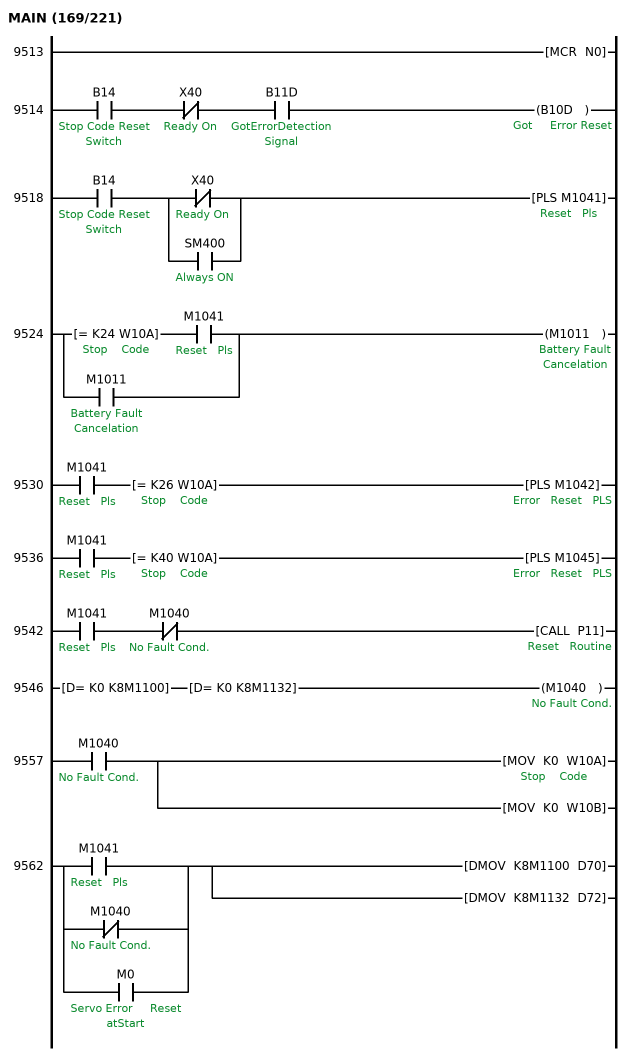
[picture p168: ladder of MAIN, rungs at steps 9513 to 9562]
9513  MCR     N0
9514  LD      B14  ; Stop Code Reset Switch
      ANI     X40  ; Ready On
      AND     B11D  ; GotErrorDetection Signal
      OUT     B10D  ; Got     Error Reset
9518  LD      B14  ; Stop Code Reset Switch
      LDI     X40  ; Ready On
      OR      SM400  ; Always ON
      ANB
      PLS     M1041  ; Reset   Pls
9524  LD=     K24 W10A  ; Stop    Code
      AND     M1041  ; Reset   Pls
      OR      M1011  ; Battery Fault   Cancelation
      OUT     M1011  ; Battery Fault   Cancelation
9530  LD      M1041  ; Reset   Pls
      AND=    K26 W10A  ; Stop    Code
      PLS     M1042  ; Error   Reset   PLS
9536  LD      M1041  ; Reset   Pls
      AND=    K40 W10A  ; Stop    Code
      PLS     M1045  ; Error   Reset   PLS
9542  LD      M1041  ; Reset   Pls
      ANI     M1040  ; No Fault Cond.
      CALL    P11  ; Reset   Routine
9546  LDD=    K0 K8M1100
      ANDD=   K0 K8M1132  ; Nozzle  Operation       Fault
      OUT     M1040  ; No Fault Cond.
9557  LD      M1040  ; No Fault Cond.
      MOV     K0 W10A
      MOV     K0 W10B
9562  LD      M1041  ; Reset   Pls
      ORI     M1040  ; No Fault Cond.
      OR      M0  ; Servo Error     Reset atStart
      DMOV    K8M1100 D70
      DMOV    K8M1132 D72
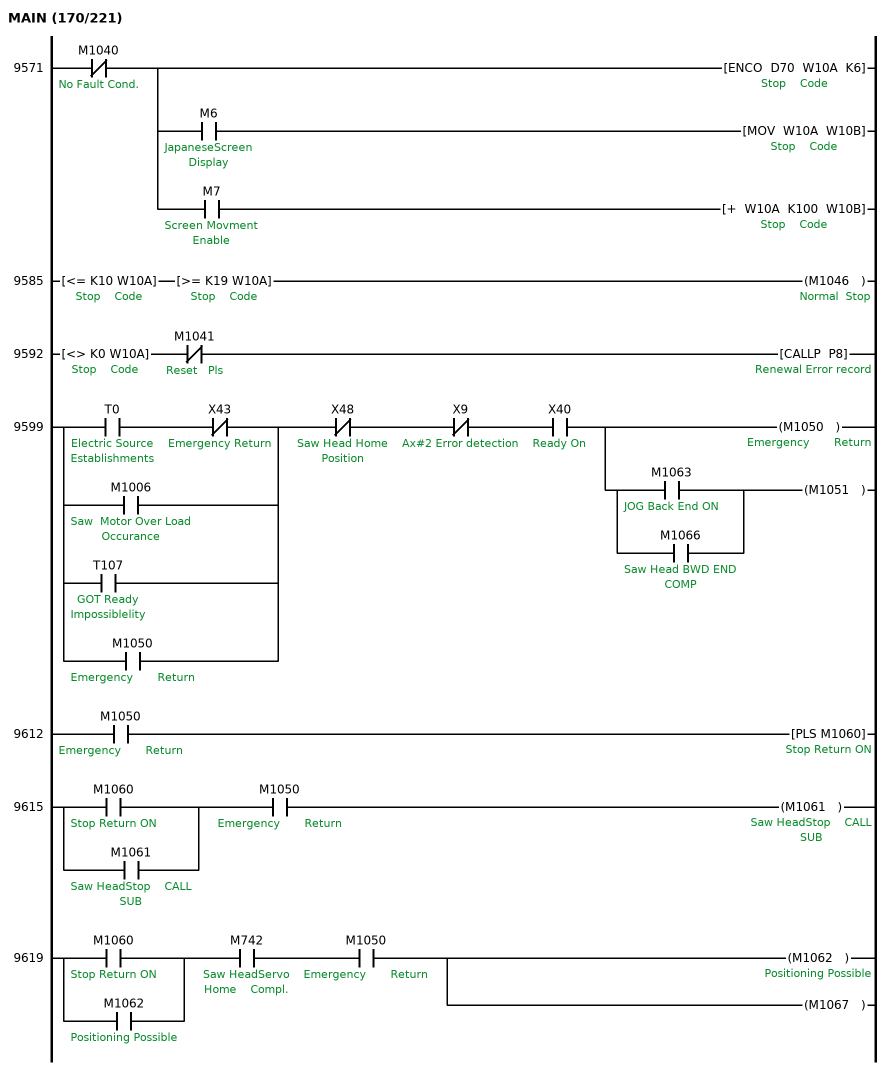
9571  LDI     M1040  ; No Fault Cond.
      ENCO    D70 W10A K6
      MPS
      AND     M6  ; JapaneseScreen Display
      MOV     W10A W10B
      MPP
      AND     M7  ; Screen Movment Enable
      +       W10A K100 W10B
9585  LD<=    K10 W10A  ; Stop    Code
      AND>=   K19 W10A  ; Stop    Code
      OUT     M1046  ; Normal  Stop
9592  LD<>    K0 W10A  ; Stop    Code
      ANI     M1041  ; Reset   Pls
      CALLP   P8  ; Renewal Error record
9599  LD      T0  ; Electric Source Establishments
      ANI     X43  ; Emergency Return
      OR      M1006  ; Saw  Motor Over Load Occurance
      OR      T107  ; GOT Ready Impossiblelity
      OR      M1050  ; Emergency       Return
      ANI     X48  ; Saw Head Home Position
      ANI     X9  ; Ax#2 Error detection
      AND     X40  ; Ready On
      OUT     M1050  ; Emergency       Return
      LD      M1063  ; JOG Back End ON
      OR      M1066  ; Saw Head BWD END COMP
      ANB
      OUT     M1051
9612  LD      M1050  ; Emergency       Return
      PLS     M1060  ; Stop Return ON
9615  LD      M1060  ; Stop Return ON
      OR      M1061  ; Saw HeadStop    CALL SUB
      AND     M1050  ; Emergency       Return
      OUT     M1061  ; Saw HeadStop    CALL SUB
9619  LD      M1060  ; Stop Return ON
      OR      M1062  ; Positioning Possible
      AND     M742  ; Saw HeadServo   Home    Compl.
      AND     M1050  ; Emergency       Return
      OUT     M1062  ; Positioning Possible
      OUT     M1067
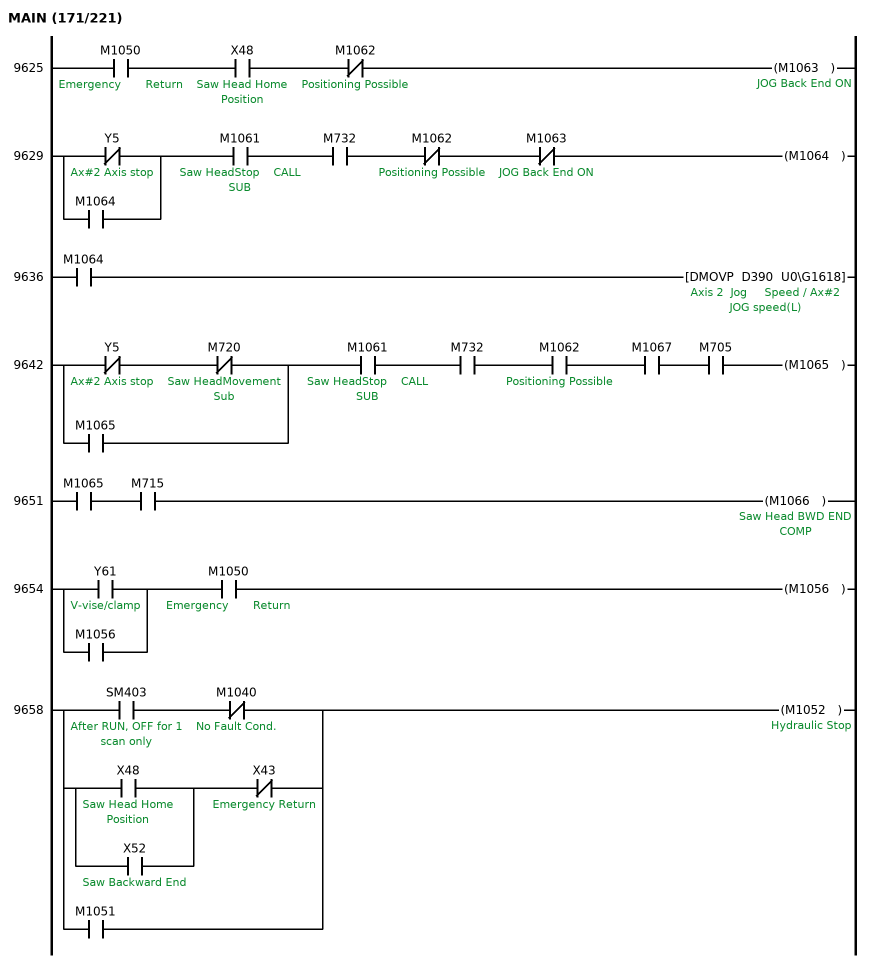
9625  LD      M1050  ; Emergency       Return
      AND     X48  ; Saw Head Home Position
      ANI     M1062  ; Positioning Possible
      OUT     M1063  ; JOG Back End ON
9629  LDI     Y5  ; Ax#2 Axis stop
      OR      M1064
      AND     M1061  ; Saw HeadStop    CALL SUB
      AND     M732
      ANI     M1062  ; Positioning Possible
      ANI     M1063  ; JOG Back End ON
      OUT     M1064
9636  LD      M1064
      DMOVP   D390 U0\G1618
9642  LDI     Y5  ; Ax#2 Axis stop
      ANI     M720  ; Saw HeadMovementSub
      OR      M1065
      AND     M1061  ; Saw HeadStop    CALL SUB
      AND     M732
      AND     M1062  ; Positioning Possible
      AND     M1067
      AND     M705
      OUT     M1065
9651  LD      M1065
      AND     M715
      OUT     M1066  ; Saw Head BWD END COMP
9654  LD      Y61  ; V-vise/clamp
      OR      M1056
      AND     M1050  ; Emergency       Return
      OUT     M1056
9658  LD      SM403  ; After RUN, OFF for 1 scan only
      ANI     M1040  ; No Fault Cond.
      LD      X48  ; Saw Head Home Position
      OR      X52  ; Saw Backward End
      ANI     X43  ; Emergency Return
      ORB
      OR      M1051
      OUT     M1052  ; Hydraulic Stop
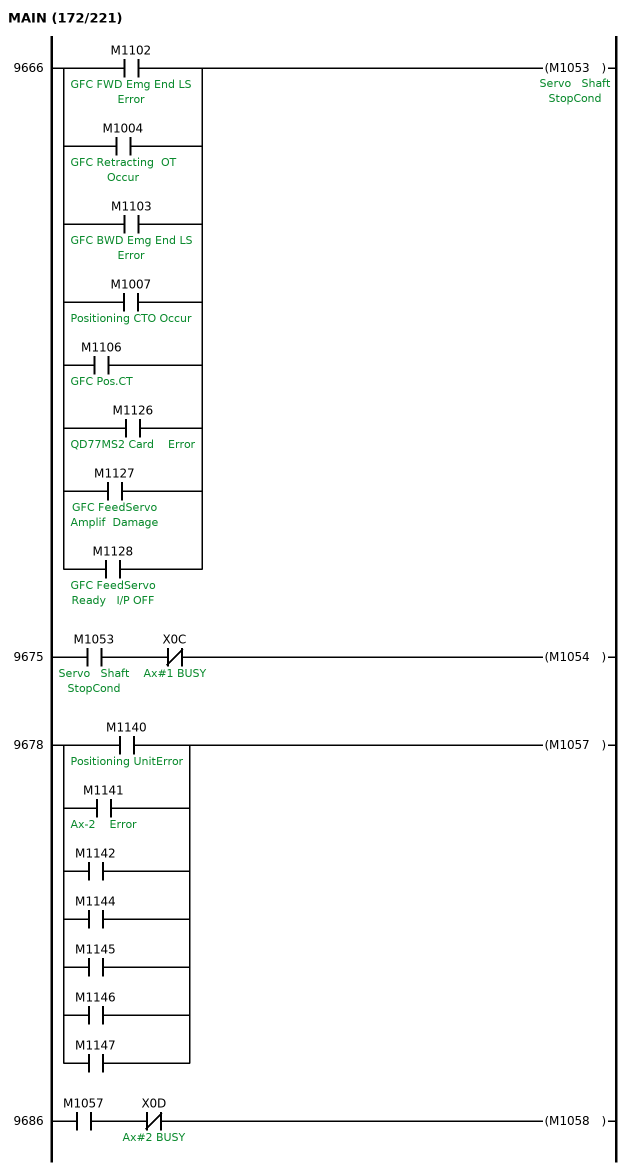
9666  LD      M1102  ; GFC FWD Emg End LS  Error
      OR      M1004  ; GFC Retracting  OT Occur
      OR      M1103  ; GFC BWD Emg End LS Error
      OR      M1007  ; Positioning CTO Occur
      OR      M1106  ; GFC Pos.CT
      OR      M1126  ; QD77MS2 Card    Error
      OR      M1127  ; GFC FeedServo   Amplif  Damage
      OR      M1128  ; GFC FeedServo   Ready   I/P OFF
      OUT     M1053  ; Servo   Shaft   StopCond
9675  LD      M1053  ; Servo   Shaft   StopCond
      ANI     X0C  ; Ax#1 BUSY
      OUT     M1054
9678  LD      M1140  ; Positioning UnitError
      OR      M1141  ; Ax-2    Error
      OR      M1142
      OR      M1144
      OR      M1145
      OR      M1146
      OR      M1147
      OUT     M1057
9686  LD      M1057
      ANI     X0D  ; Ax#2 BUSY
      OUT     M1058
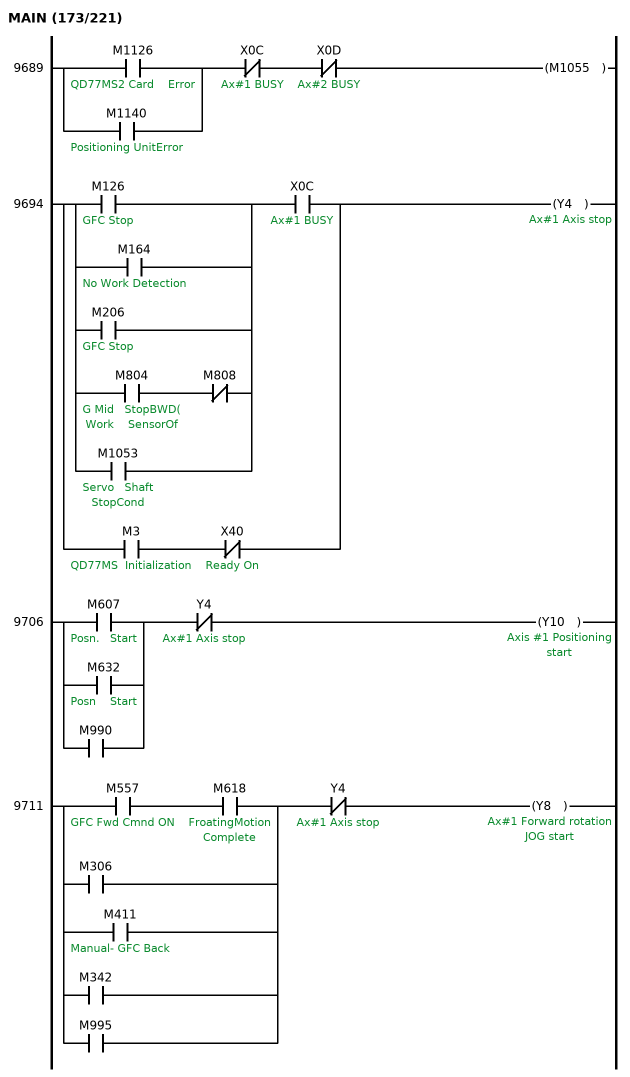
9689  LD      M1126  ; QD77MS2 Card    Error
      OR      M1140  ; Positioning UnitError
      ANI     X0C  ; Ax#1 BUSY
      ANI     X0D  ; Ax#2 BUSY
      OUT     M1055
9694  LD      M126  ; GFC Stop
      OR      M164  ; No Work Detection
      OR      M206  ; GFC Stop
      LD      M804  ; G Mid   StopBWD(Work    SensorOf
      ANI     M808
      ORB
      OR      M1053  ; Servo   Shaft   StopCond
      AND     X0C  ; Ax#1 BUSY
      LD      M3  ; QD77MS  Initialization
      ANI     X40  ; Ready On
      ORB
      OUT     Y4  ; Ax#1 Axis stop
9706  LD      M607  ; Posn.   Start
      OR      M632  ; Posn    Start
      OR      M990
      ANI     Y4  ; Ax#1 Axis stop
      OUT     Y10  ; Axis #1 Positioning start
9711  LD      M557  ; GFC Fwd Cmnd ON
      AND     M618  ; FroatingMotion  Complete
      OR      M306
      OR      M411  ; Manual- GFC Back
      OR      M342
      OR      M995
      ANI     Y4  ; Ax#1 Axis stop
      OUT     Y8  ; Ax#1 Forward rotation JOG start
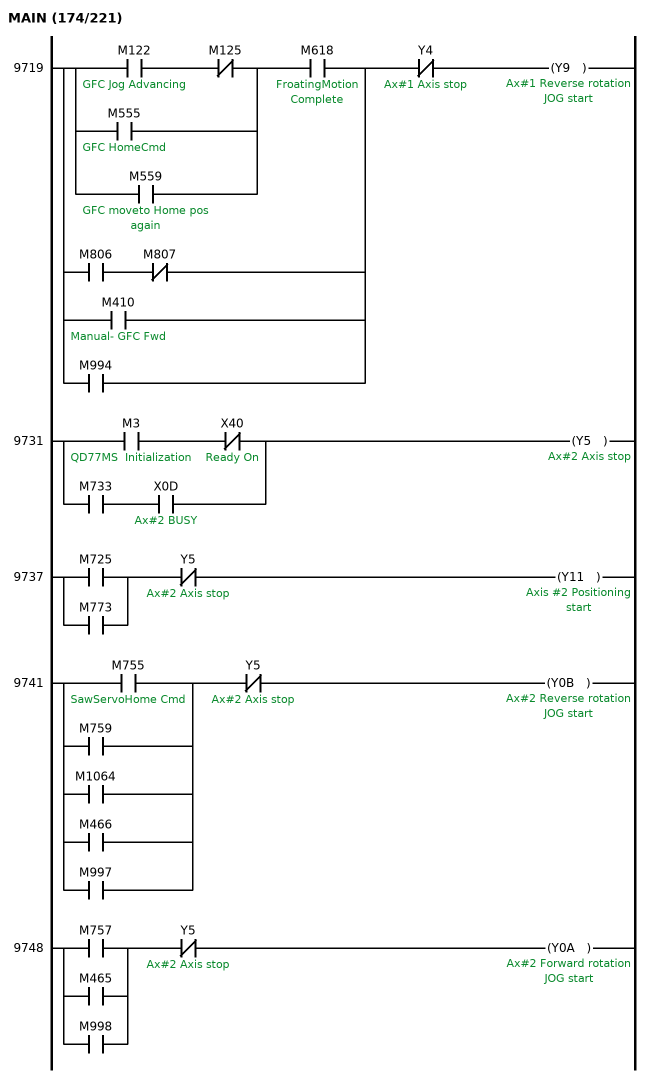
9719  LD      M122  ; GFC Jog Advancing
      ANI     M125
      OR      M555  ; GFC HomeCmd
      OR      M559  ; GFC moveto Home pos     again
      AND     M618  ; FroatingMotion  Complete
      LD      M806
      ANI     M807
      ORB
      OR      M410  ; Manual- GFC Fwd
      OR      M994
      ANI     Y4  ; Ax#1 Axis stop
      OUT     Y9  ; Ax#1 Reverse rotation JOG start
9731  LD      M3  ; QD77MS  Initialization
      ANI     X40  ; Ready On
      LD      M733
      AND     X0D  ; Ax#2 BUSY
      ORB
      OUT     Y5  ; Ax#2 Axis stop
9737  LD      M725
      OR      M773
      ANI     Y5  ; Ax#2 Axis stop
      OUT     Y11  ; Axis #2 Positioning start
9741  LD      M755  ; SawServoHome Cmd
      OR      M759
      OR      M1064
      OR      M466
      OR      M997
      ANI     Y5  ; Ax#2 Axis stop
      OUT     Y0B  ; Ax#2 Reverse rotation JOG start
9748  LD      M757
      OR      M465
      OR      M998
      ANI     Y5  ; Ax#2 Axis stop
      OUT     Y0A  ; Ax#2 Forward rotation JOG start
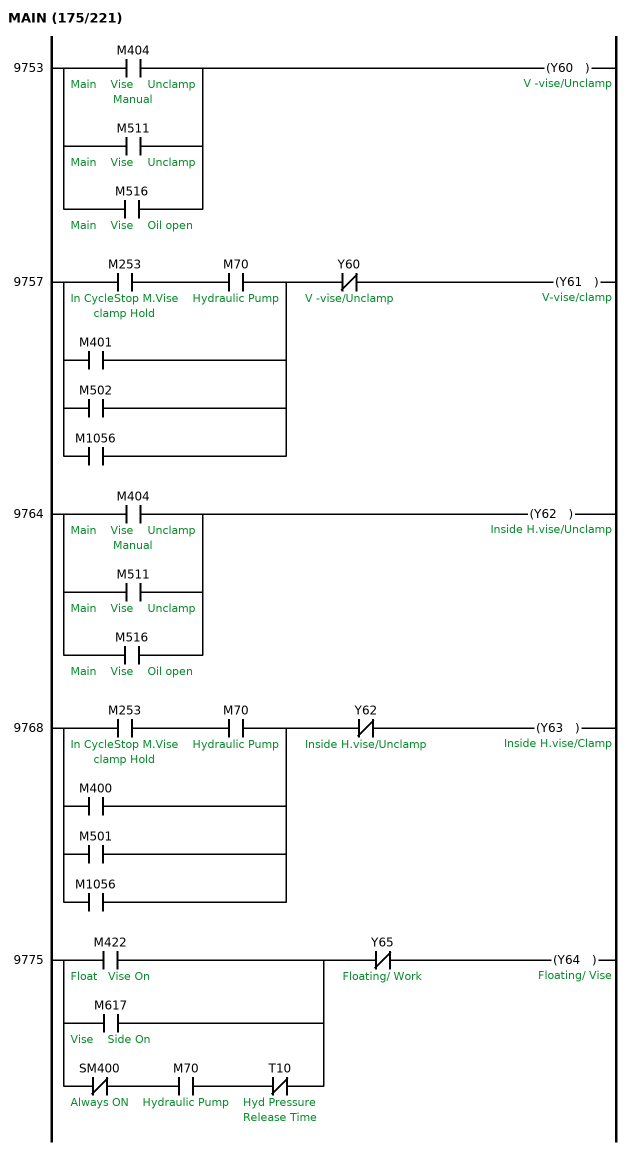
9753  LD      M404  ; Main    Vise    Unclamp Manual
      OR      M511  ; Main    Vise    Unclamp
      OR      M516  ; Main    Vise    Oil open
      OUT     Y60  ; V -vise/Unclamp
9757  LD      M253  ; In CycleStop M.Vise clamp Hold
      AND     M70  ; Hydraulic Pump
      OR      M401
      OR      M502
      OR      M1056
      ANI     Y60  ; V -vise/Unclamp
      OUT     Y61  ; V-vise/clamp
9764  LD      M404  ; Main    Vise    Unclamp Manual
      OR      M511  ; Main    Vise    Unclamp
      OR      M516  ; Main    Vise    Oil open
      OUT     Y62  ; Inside H.vise/Unclamp
9768  LD      M253  ; In CycleStop M.Vise clamp Hold
      AND     M70  ; Hydraulic Pump
      OR      M400
      OR      M501
      OR      M1056
      ANI     Y62  ; Inside H.vise/Unclamp
      OUT     Y63  ; Inside H.vise/Clamp
9775  LD      M422  ; Float   Vise On
      OR      M617  ; Vise    Side On
      LDI     SM400  ; Always ON
      AND     M70  ; Hydraulic Pump
      ANI     T10  ; Hyd Pressure    Release Time
      ORB
      ANI     Y65  ; Floating/ Work
      OUT     Y64  ; Floating/ Vise
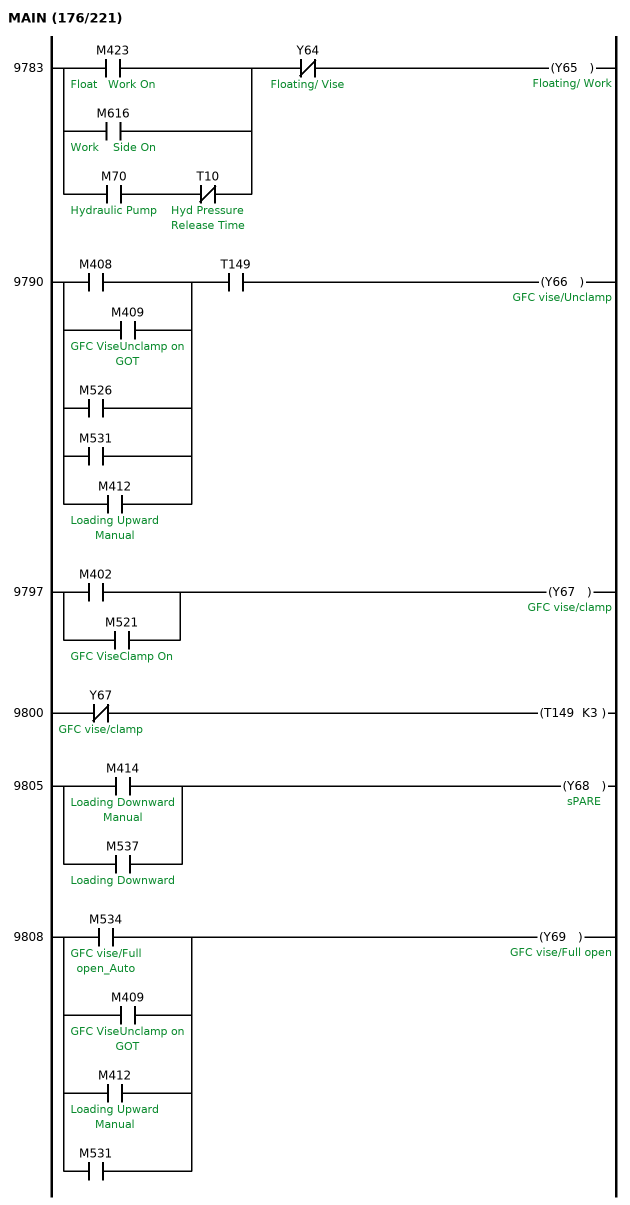
9783  LD      M423  ; Float   Work On
      OR      M616  ; Work    Side On
      LD      M70  ; Hydraulic Pump
      ANI     T10  ; Hyd Pressure    Release Time
      ORB
      ANI     Y64  ; Floating/ Vise
      OUT     Y65  ; Floating/ Work
9790  LD      M408
      OR      M409  ; GFC ViseUnclamp on GOT
      OR      M526
      OR      M531
      OR      M412  ; Loading Upward  Manual
      AND     T149
      OUT     Y66  ; GFC vise/Unclamp
9797  LD      M402
      OR      M521  ; GFC ViseClamp On
      OUT     Y67  ; GFC vise/clamp
9800  LDI     Y67  ; GFC vise/clamp
      OUT     T149 K3
9805  LD      M414  ; Loading Downward Manual
      OR      M537  ; Loading Downward
      OUT     Y68  ; sPARE
9808  LD      M534  ; GFC vise/Full open_Auto
      OR      M409  ; GFC ViseUnclamp on GOT
      OR      M412  ; Loading Upward  Manual
      OR      M531
      OUT     Y69  ; GFC vise/Full open
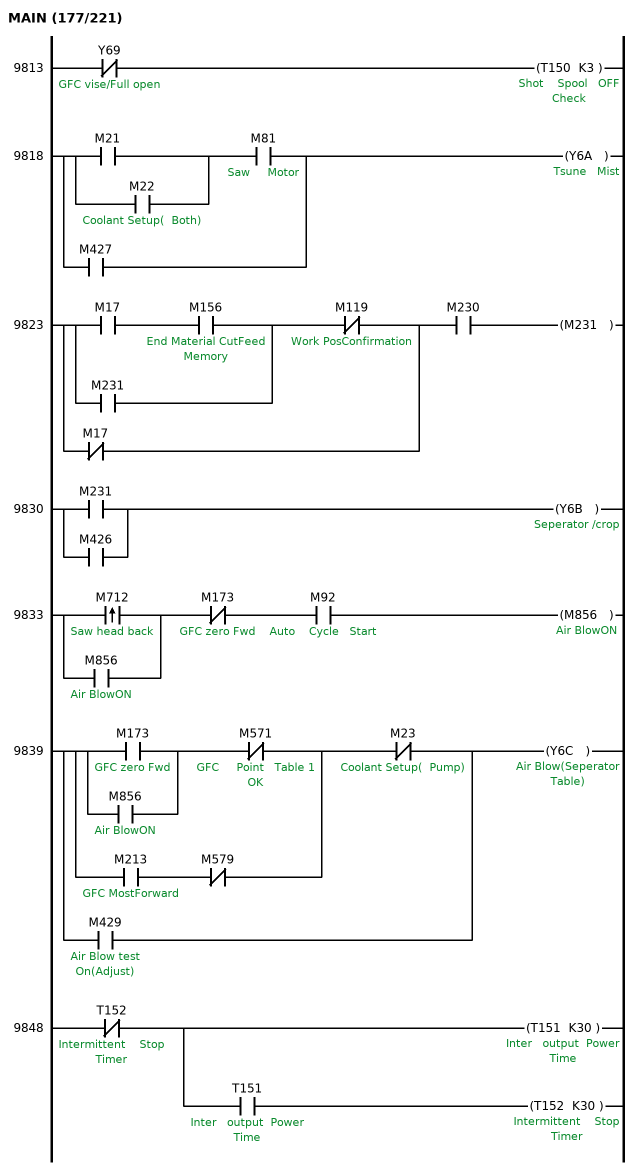
9813  LDI     Y69  ; GFC vise/Full open
      OUT     T150 K3  ; Shot    Spool   OFF     Check
9818  LD      M21
      OR      M22  ; Coolant Setup(  Both)
      AND     M81  ; Saw     Motor
      OR      M427
      OUT     Y6A  ; Tsune   Mist
9823  LD      M17
      AND     M156  ; End Material CutFeed Memory
      OR      M231
      ANI     M119  ; Work PosConfirmation
      ORI     M17
      AND     M230
      OUT     M231
9830  LD      M231
      OR      M426
      OUT     Y6B  ; Seperator /crop
9833  LDP     M712  ; Saw head back
      OR      M856  ; Air BlowON
      ANI     M173  ; GFC zero Fwd
      AND     M92  ; Auto    Cycle   Start
      OUT     M856  ; Air BlowON
9839  LD      M173  ; GFC zero Fwd
      OR      M856  ; Air BlowON
      ANI     M571  ; GFC     Point   Table 1 OK
      LD      M213  ; GFC MostForward
      ANI     M579
      ORB
      ANI     M23  ; Coolant Setup(  Pump)
      OR      M429  ; Air Blow test On(Adjust)
      OUT     Y6C  ; Air Blow(Seperator Table)
9848  LDI     T152  ; Intermittent    Stop    Timer
      OUT     T151 K30  ; Inter   output  Power   Time
      AND     T151  ; Inter   output  Power   Time
      OUT     T152 K30  ; Intermittent    Stop    Timer
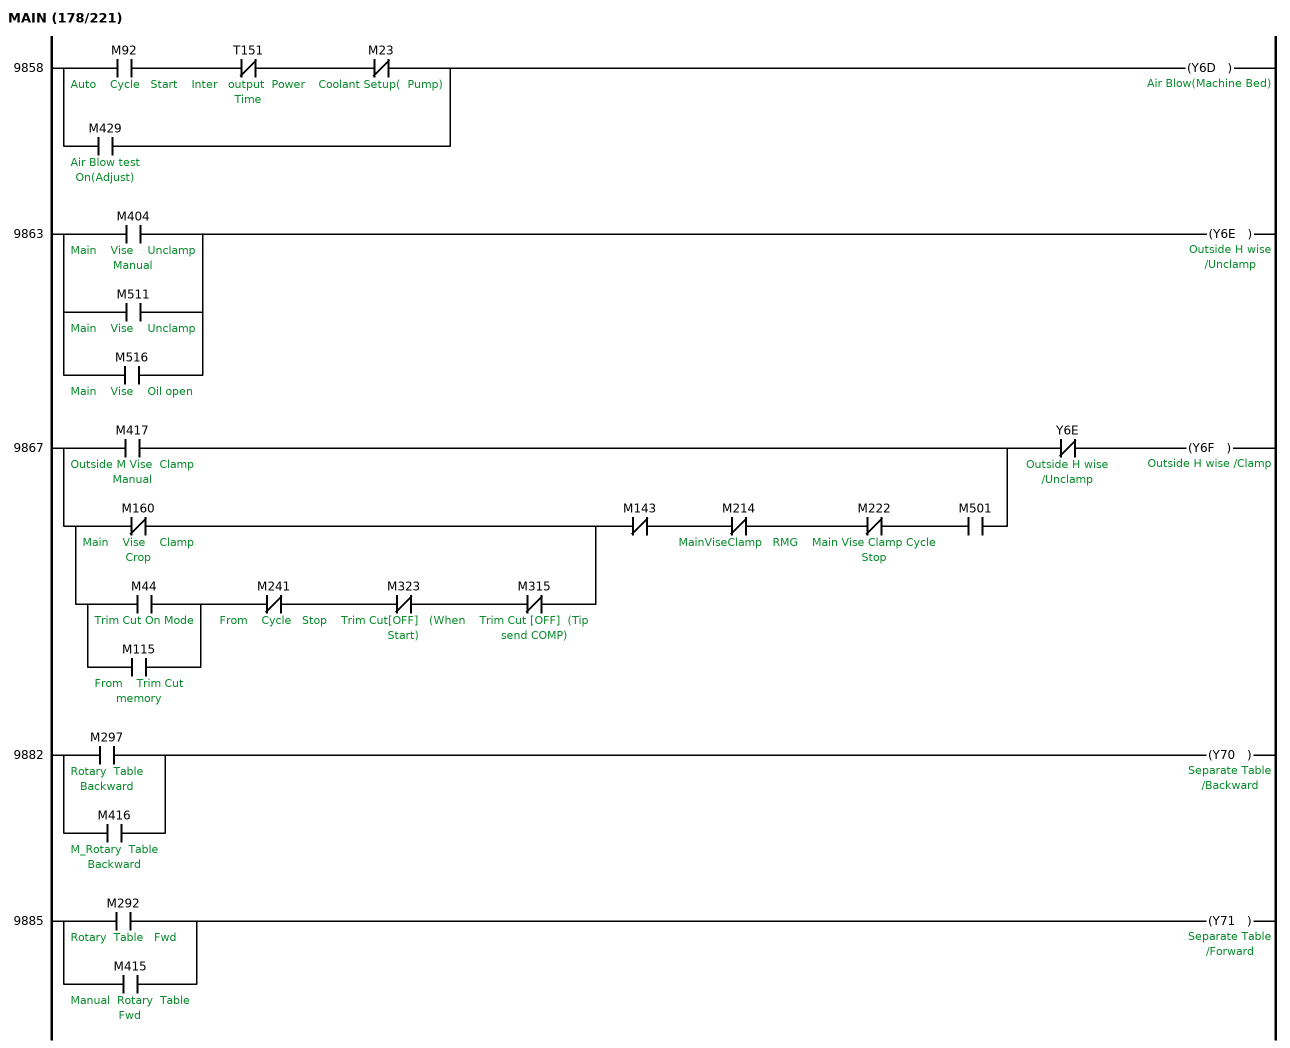
9858  LD      M92  ; Auto    Cycle   Start
      ANI     T151  ; Inter   output  Power   Time
      ANI     M23  ; Coolant Setup(  Pump)
      OR      M429  ; Air Blow test On(Adjust)
      OUT     Y6D  ; Air Blow(Machine Bed)
9863  LD      M404  ; Main    Vise    Unclamp Manual
      OR      M511  ; Main    Vise    Unclamp
      OR      M516  ; Main    Vise    Oil open
      OUT     Y6E  ; Outside H wise /Unclamp
9867  LD      M417  ; Outside M Vise  Clamp   Manual
      LDI     M160  ; Main    Vise    Clamp   Crop
      LD      M44  ; Trim Cut On Mode
      OR      M115  ; From    Trim Cut memory
      ANI     M241  ; From    Cycle   Stop
      ANI     M323  ; Trim Cut[OFF]   (When   Start)
      ANI     M315  ; Trim Cut [OFF]  (Tip send COMP)
      ORB
      ANI     M143
      ANI     M214  ; MainViseClamp   RMG
      ANI     M222  ; Main Vise Clamp Cycle Stop
      AND     M501
      ORB
      ANI     Y6E  ; Outside H wise /Unclamp
      OUT     Y6F  ; Outside H wise /Clamp
9882  LD      M297  ; Rotary  Table   Backward
      OR      M416  ; M_Rotary  Table Backward
      OUT     Y70  ; Separate Table /Backward
9885  LD      M292  ; Rotary  Table   Fwd
      OR      M415  ; Manual  Rotary  Table   Fwd
      OUT     Y71  ; Separate Table /Forward
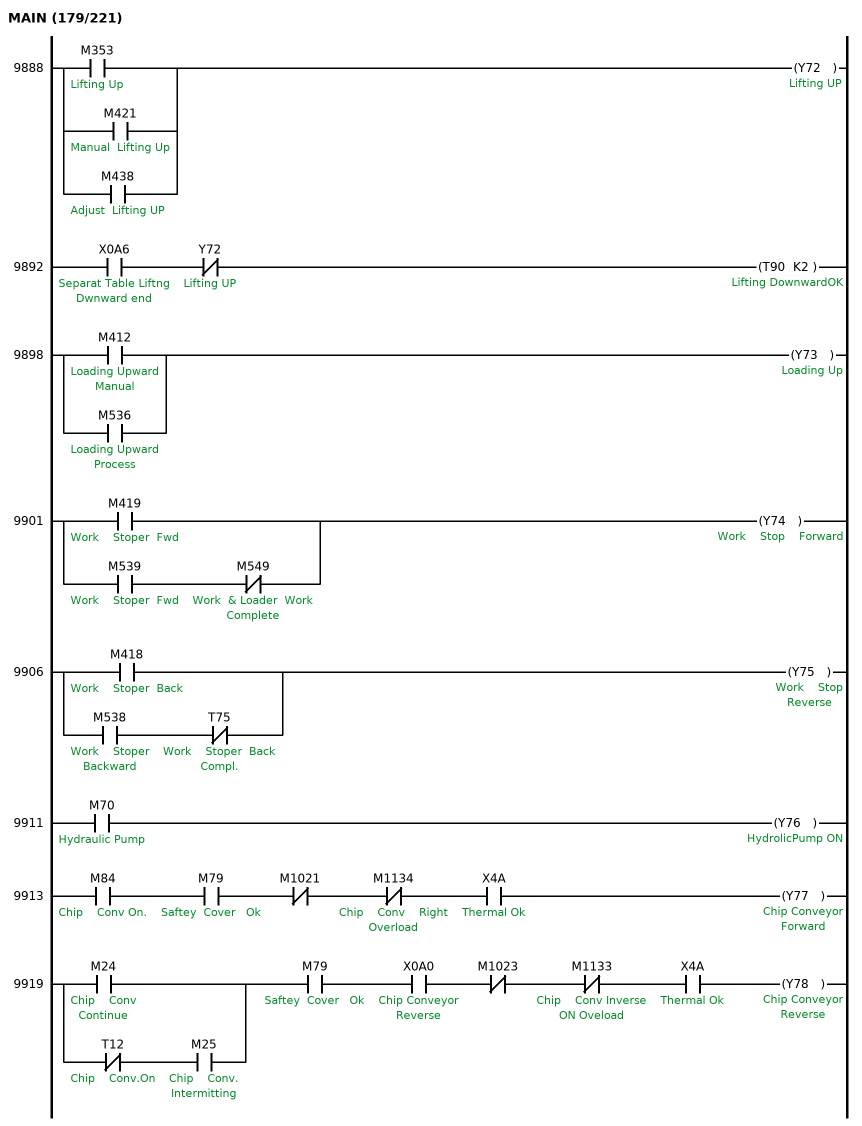
9888  LD      M353  ; Lifting Up
      OR      M421  ; Manual  Lifting Up
      OR      M438  ; Adjust  Lifting UP
      OUT     Y72  ; Lifting UP
9892  LD      X0A6  ; Separat Table Liftng Dwnward end
      ANI     Y72  ; Lifting UP
      OUT     T90 K2  ; Lifting DownwardOK
9898  LD      M412  ; Loading Upward  Manual
      OR      M536  ; Loading Upward  Process
      OUT     Y73  ; Loading Up
9901  LD      M419  ; Work    Stoper  Fwd
      LD      M539  ; Work    Stoper  Fwd
      ANI     M549  ; Work  & Loader  Work Complete
      ORB
      OUT     Y74  ; Work    Stop    Forward
9906  LD      M418  ; Work    Stoper  Back
      LD      M538  ; Work    Stoper  Backward
      ANI     T75  ; Work    Stoper  Back    Compl.
      ORB
      OUT     Y75  ; Work    Stop    Reverse
9911  LD      M70  ; Hydraulic Pump
      OUT     Y76  ; HydrolicPump ON
9913  LD      M84  ; Chip    Conv On.
      AND     M79  ; Saftey  Cover   Ok
      ANI     M1021
      ANI     M1134  ; Chip    Conv    Right   Overload
      AND     X4A  ; Thermal Ok
      OUT     Y77  ; Chip Conveyor Forward
9919  LD      M24  ; Chip    Conv    Continue
      LDI     T12  ; Chip    Conv.On
      AND     M25  ; Chip    Conv.   Intermitting
      ORB
      AND     M79  ; Saftey  Cover   Ok
      AND     X0A0  ; Chip Conveyor Reverse
      ANI     M1023
      ANI     M1133  ; Chip    Conv Inverse ON Oveload
      AND     X4A  ; Thermal Ok
      OUT     Y78  ; Chip Conveyor Reverse
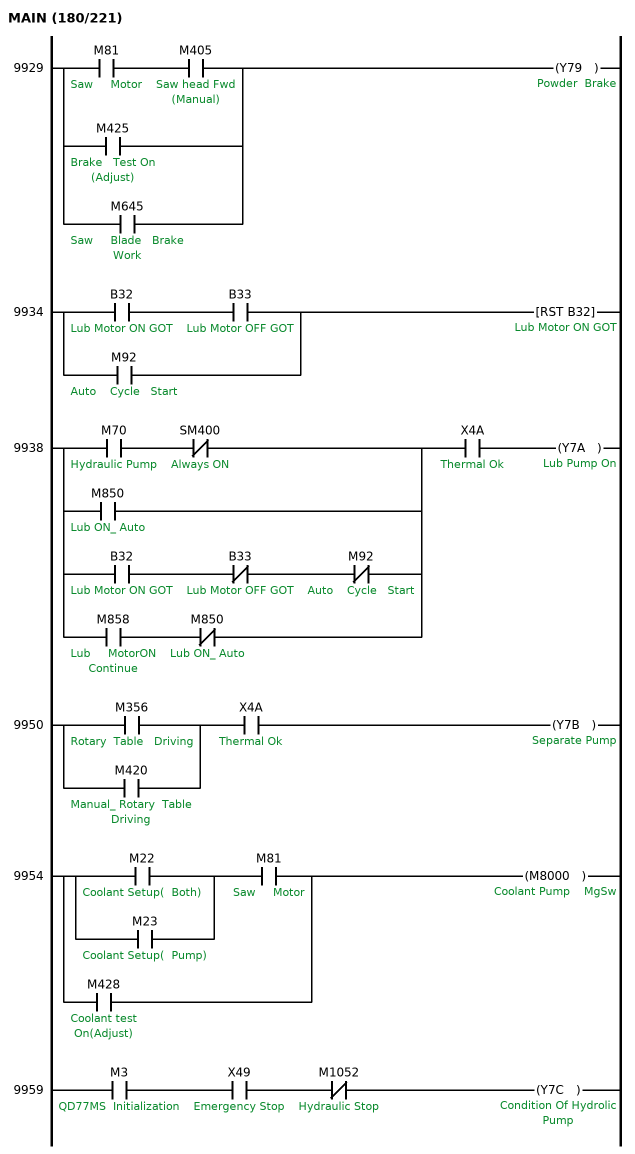
9929  LD      M81  ; Saw     Motor
      AND     M405  ; Saw head Fwd    (Manual)
      OR      M425  ; Brake   Test On (Adjust)
      OR      M645  ; Saw     Blade   Brake   Work
      OUT     Y79  ; Powder  Brake
9934  LD      B32  ; Lub Motor ON GOT
      AND     B33  ; Lub Motor OFF GOT
      OR      M92  ; Auto    Cycle   Start
      RST     B32  ; Lub Motor ON GOT
9938  LD      M70  ; Hydraulic Pump
      ANI     SM400  ; Always ON
      OR      M850  ; Lub ON_ Auto
      LD      B32  ; Lub Motor ON GOT
      ANI     B33  ; Lub Motor OFF GOT
      ANI     M92  ; Auto    Cycle   Start
      ORB
      LD      M858  ; Lub     MotorON Continue
      ANI     M850  ; Lub ON_ Auto
      ORB
      AND     X4A  ; Thermal Ok
      OUT     Y7A  ; Lub Pump On
9950  LD      M356  ; Rotary  Table   Driving
      OR      M420  ; Manual_ Rotary  Table   Driving
      AND     X4A  ; Thermal Ok
      OUT     Y7B  ; Separate Pump
9954  LD      M22  ; Coolant Setup(  Both)
      OR      M23  ; Coolant Setup(  Pump)
      AND     M81  ; Saw     Motor
      OR      M428  ; Coolant test On(Adjust)
      OUT     M8000  ; Coolant Pump    MgSw
9959  LD      M3  ; QD77MS  Initialization
      AND     X49  ; Emergency Stop
      ANI     M1052  ; Hydraulic Stop
      OUT     Y7C  ; Condition Of Hydrolic Pump
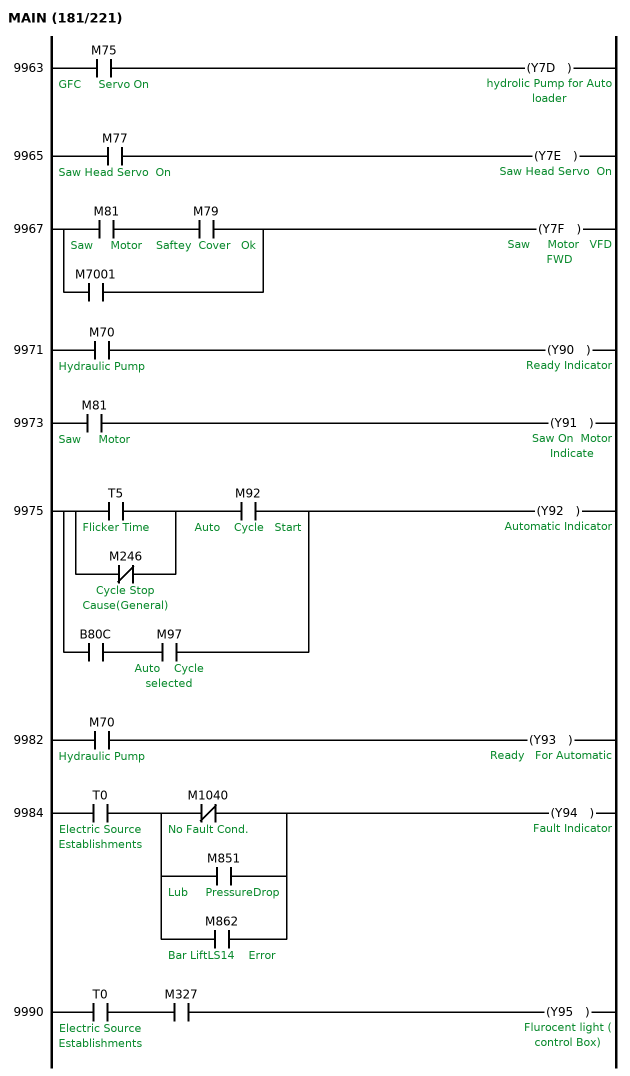
9963  LD      M75  ; GFC     Servo On
      OUT     Y7D  ; hydrolic Pump for Auto loader
9965  LD      M77  ; Saw Head Servo  On
      OUT     Y7E  ; Saw Head Servo  On
9967  LD      M81  ; Saw     Motor
      AND     M79  ; Saftey  Cover   Ok
      OR      M7001
      OUT     Y7F  ; Saw     Motor   VFD FWD
9971  LD      M70  ; Hydraulic Pump
      OUT     Y90  ; Ready Indicator
9973  LD      M81  ; Saw     Motor
      OUT     Y91  ; Saw On  Motor   Indicate
9975  LD      T5  ; Flicker Time
      ORI     M246  ; Cycle Stop Cause(General)
      AND     M92  ; Auto    Cycle   Start
      LD      B80C
      AND     M97  ; Auto    Cycle   selected
      ORB
      OUT     Y92  ; Automatic Indicator
9982  LD      M70  ; Hydraulic Pump
      OUT     Y93  ; Ready   For Automatic
9984  LD      T0  ; Electric Source Establishments
      LDI     M1040  ; No Fault Cond.
      OR      M851  ; Lub     PressureDrop
      OR      M862  ; Bar LiftLS14    Error
      ANB
      OUT     Y94  ; Fault Indicator
9990  LD      T0  ; Electric Source Establishments
      AND     M327
      OUT     Y95  ; Flurocent light ( control Box)
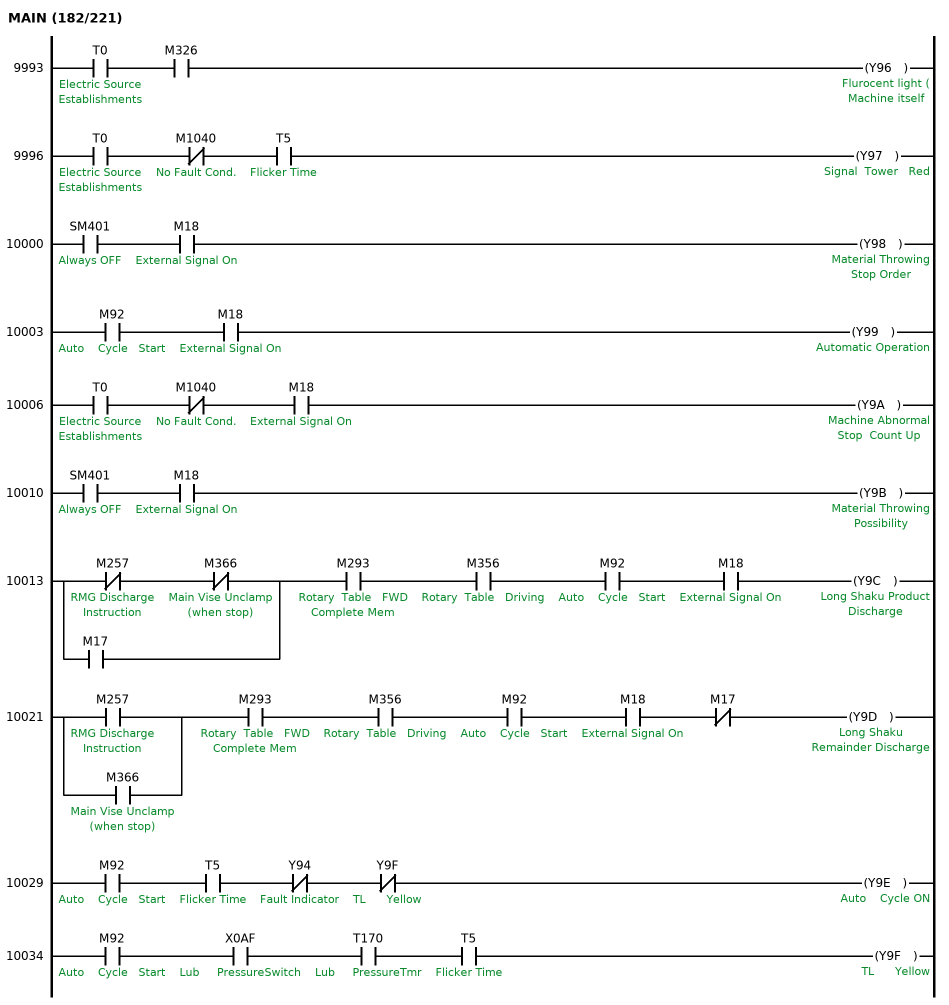
9993  LD      T0  ; Electric Source Establishments
      AND     M326
      OUT     Y96  ; Flurocent light ( Machine itself
9996  LD      T0  ; Electric Source Establishments
      ANI     M1040  ; No Fault Cond.
      AND     T5  ; Flicker Time
      OUT     Y97  ; Signal  Tower   Red
10000 LD      SM401  ; Always OFF
      AND     M18  ; External Signal On
      OUT     Y98  ; Material Throwing Stop Order
10003 LD      M92  ; Auto    Cycle   Start
      AND     M18  ; External Signal On
      OUT     Y99  ; Automatic Operation
10006 LD      T0  ; Electric Source Establishments
      ANI     M1040  ; No Fault Cond.
      AND     M18  ; External Signal On
      OUT     Y9A  ; Machine Abnormal Stop  Count Up
10010 LD      SM401  ; Always OFF
      AND     M18  ; External Signal On
      OUT     Y9B  ; Material Throwing Possibility
10013 LDI     M257  ; RMG Discharge Instruction
      ANI     M366  ; Main Vise Unclamp (when stop)
      OR      M17
      AND     M293  ; Rotary  Table   FWD Complete Mem
      AND     M356  ; Rotary  Table   Driving
      AND     M92  ; Auto    Cycle   Start
      AND     M18  ; External Signal On
      OUT     Y9C  ; Long Shaku Product Discharge
10021 LD      M257  ; RMG Discharge Instruction
      OR      M366  ; Main Vise Unclamp (when stop)
      AND     M293  ; Rotary  Table   FWD Complete Mem
      AND     M356  ; Rotary  Table   Driving
      AND     M92  ; Auto    Cycle   Start
      AND     M18  ; External Signal On
      ANI     M17
      OUT     Y9D  ; Long Shaku Remainder Discharge
10029 LD      M92  ; Auto    Cycle   Start
      AND     T5  ; Flicker Time
      ANI     Y94  ; Fault Indicator
      ANI     Y9F  ; TL      Yellow
      OUT     Y9E  ; Auto    Cycle ON
10034 LD      M92  ; Auto    Cycle   Start
      AND     X0AF  ; Lub     PressureSwitch
      AND     T170  ; Lub     PressureTmr
      AND     T5  ; Flicker Time
      OUT     Y9F  ; TL      Yellow
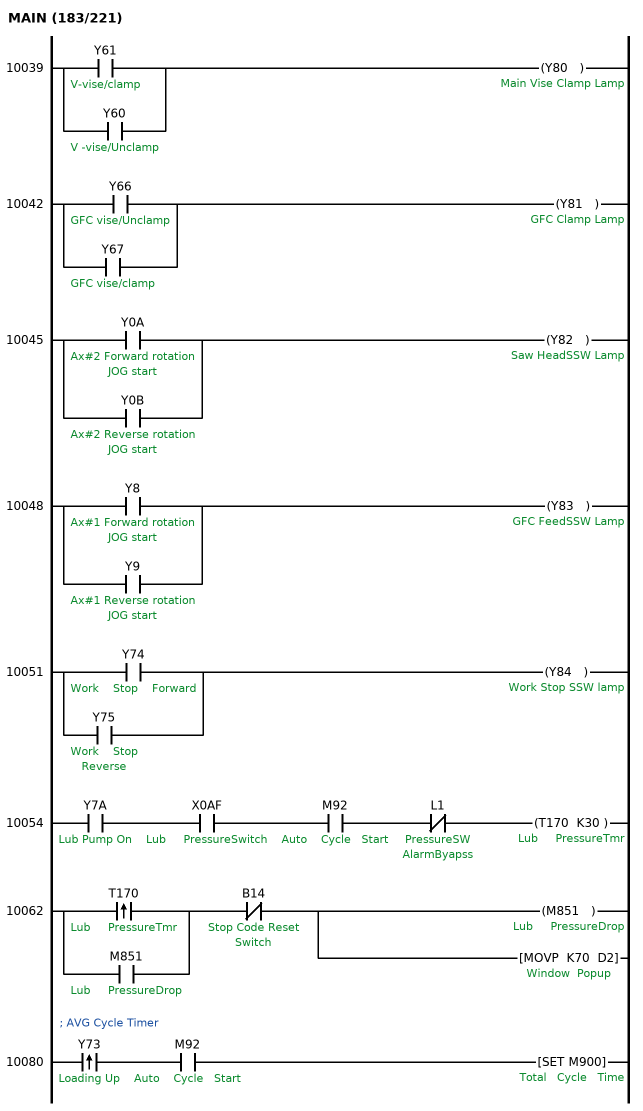
10039 LD      Y61  ; V-vise/clamp
      OR      Y60  ; V -vise/Unclamp
      OUT     Y80  ; Main Vise Clamp Lamp
10042 LD      Y66  ; GFC vise/Unclamp
      OR      Y67  ; GFC vise/clamp
      OUT     Y81  ; GFC Clamp Lamp
10045 LD      Y0A  ; Ax#2 Forward rotation JOG start
      OR      Y0B  ; Ax#2 Reverse rotation JOG start
      OUT     Y82  ; Saw HeadSSW Lamp
10048 LD      Y8  ; Ax#1 Forward rotation JOG start
      OR      Y9  ; Ax#1 Reverse rotation JOG start
      OUT     Y83  ; GFC FeedSSW Lamp
10051 LD      Y74  ; Work    Stop    Forward
      OR      Y75  ; Work    Stop    Reverse
      OUT     Y84  ; Work Stop SSW lamp
10054 LD      Y7A  ; Lub Pump On
      AND     X0AF  ; Lub     PressureSwitch
      AND     M92  ; Auto    Cycle   Start
      ANI     L1  ; PressureSW AlarmByapss
      OUT     T170 K30  ; Lub     PressureTmr
10062 LDP     T170  ; Lub     PressureTmr
      OR      M851  ; Lub     PressureDrop
      ANI     B14  ; Stop Code Reset Switch
      OUT     M851  ; Lub     PressureDrop
      MOVP    K70 D2
; AVG Cycle Timer
10080 LDP     Y73  ; Loading Up
      AND     M92  ; Auto    Cycle   Start
      SET     M900  ; Total   Cycle   Time
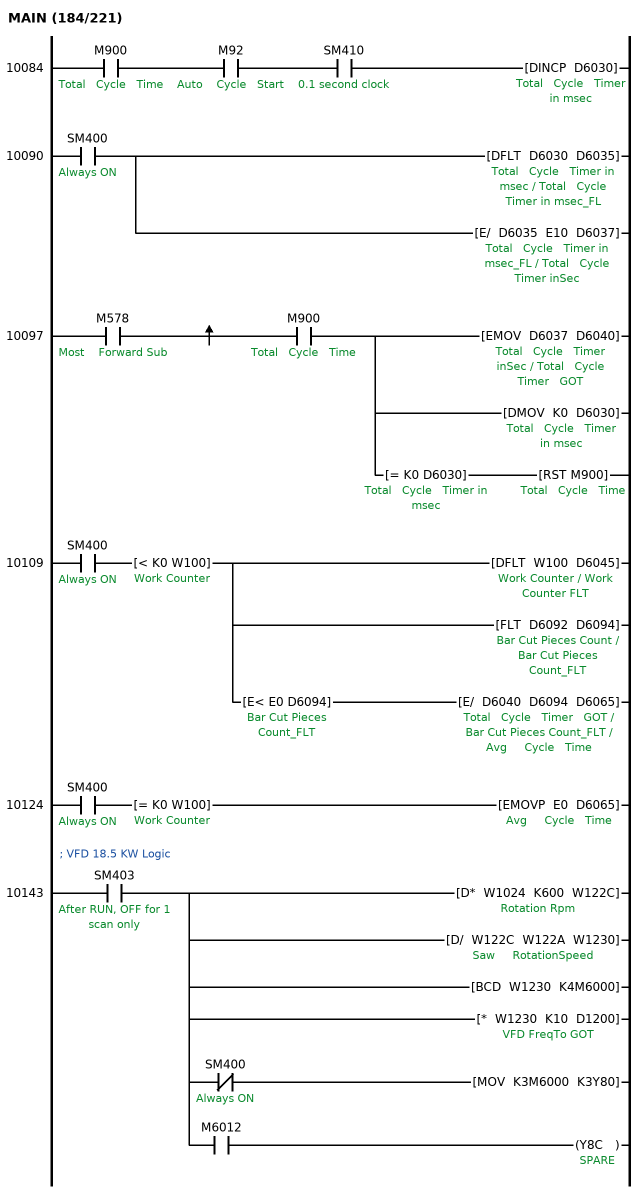
10084 LD      M900  ; Total   Cycle   Time
      AND     M92  ; Auto    Cycle   Start
      AND     SM410  ; 0.1 second clock
      DINCP   D6030  ; Total   Cycle   Timer in msec
10090 LD      SM400  ; Always ON
      DFLT    D6030 D6035  ; Total   Cycle   Timer in msec_FL
      E/      D6035 E10 D6037  ; Total   Cycle   Timer inSec
10097 LD      M578  ; Most    Forward Sub
      MEP
      AND     M900  ; Total   Cycle   Time
      EMOV    D6037 D6040  ; Total   Cycle   Timer   GOT
      DMOV    K0 D6030
      AND=    K0 D6030  ; Total   Cycle   Timer in msec
      RST     M900  ; Total   Cycle   Time
10109 LD      SM400  ; Always ON
      AND<    K0 W100  ; Work Counter
      DFLT    W100 D6045  ; Work    Counter FLT
      FLT     D6092 D6094  ; Bar Cut Pieces Count_FLT
      ANDE<   E0 D6094  ; Bar Cut Pieces Count_FLT
      E/      D6040 D6094 D6065  ; Avg     Cycle   Time
10124 LD      SM400  ; Always ON
      AND=    K0 W100  ; Work Counter
      EMOVP   E0 D6065
; VFD 18.5 KW Logic
10143 LD      SM403  ; After RUN, OFF for 1 scan only
      D*      W1024 K600 W122C
      D/      W122C W122A W1230  ; Saw     RotationSpeed
      BCD     W1230 K4M6000
      *       W1230 K10 D1200  ; VFD FreqTo GOT
      MPS
      ANI     SM400  ; Always ON
      MOV     K3M6000 K3Y80
      MPP
      AND     M6012
      OUT     Y8C  ; SPARE
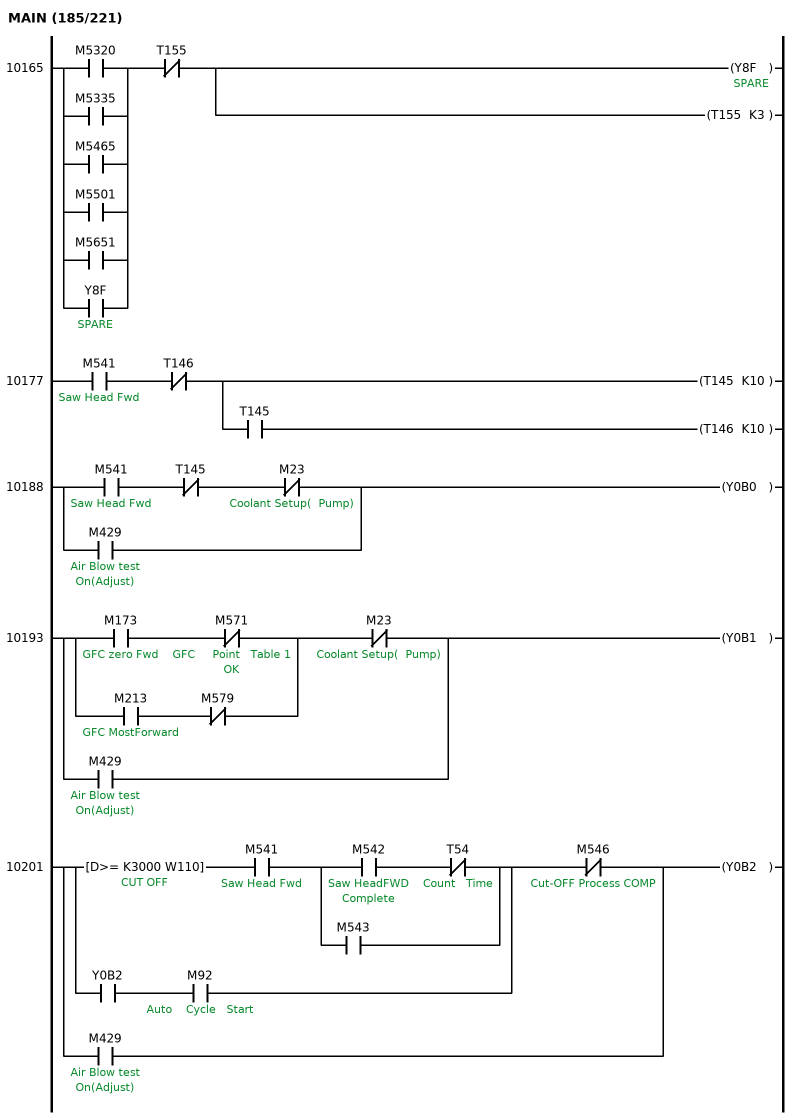
10165 LD      M5320
      OR      M5335
      OR      M5465
      OR      M5501
      OR      M5651
      OR      Y8F  ; SPARE
      ANI     T155
      OUT     Y8F  ; SPARE
      OUT     T155 K3
10177 LD      M541  ; Saw Head Fwd
      ANI     T146
      OUT     T145 K10
      AND     T145
      OUT     T146 K10
10188 LD      M541  ; Saw Head Fwd
      ANI     T145
      ANI     M23  ; Coolant Setup(  Pump)
      OR      M429  ; Air Blow test On(Adjust)
      OUT     Y0B0
10193 LD      M173  ; GFC zero Fwd
      ANI     M571  ; GFC     Point   Table 1 OK
      LD      M213  ; GFC MostForward
      ANI     M579
      ORB
      ANI     M23  ; Coolant Setup(  Pump)
      OR      M429  ; Air Blow test On(Adjust)
      OUT     Y0B1
10201 LDD>=   K3000 W110  ; CUT OFF
      AND     M541  ; Saw Head Fwd
      LD      M542  ; Saw HeadFWD     Complete
      ANI     T54  ; Count   Time
      OR      M543
      ANB
      LD      Y0B2
      AND     M92  ; Auto    Cycle   Start
      ORB
      ANI     M546  ; Cut-OFF Process COMP
      OR      M429  ; Air Blow test On(Adjust)
      OUT     Y0B2
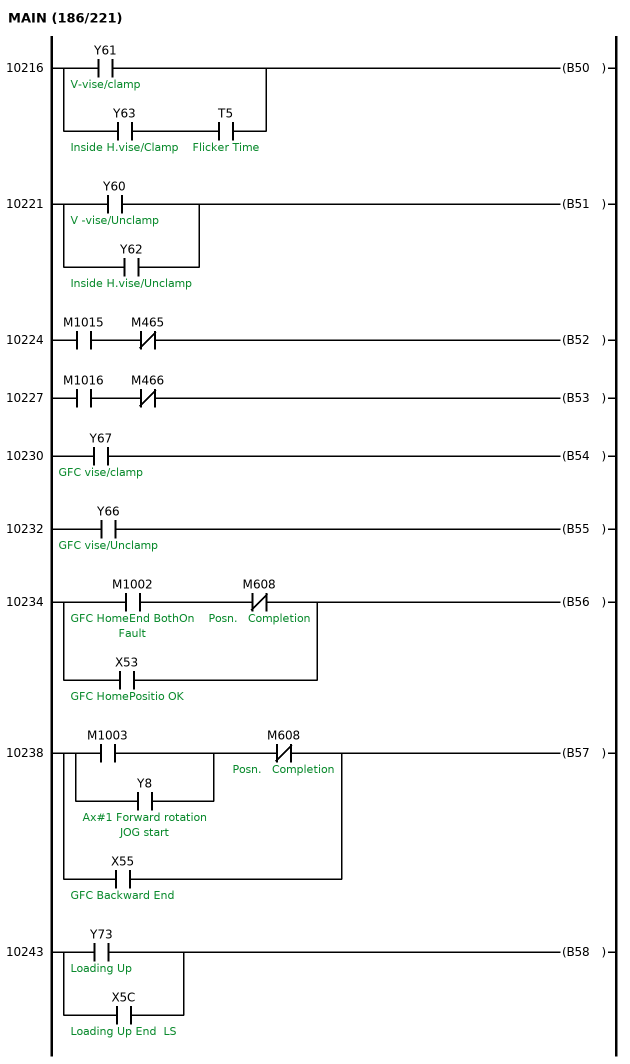
10216 LD      Y61  ; V-vise/clamp
      LD      Y63  ; Inside H.vise/Clamp
      AND     T5  ; Flicker Time
      ORB
      OUT     B50
10221 LD      Y60  ; V -vise/Unclamp
      OR      Y62  ; Inside H.vise/Unclamp
      OUT     B51
10224 LD      M1015
      ANI     M465
      OUT     B52
10227 LD      M1016
      ANI     M466
      OUT     B53
10230 LD      Y67  ; GFC vise/clamp
      OUT     B54
10232 LD      Y66  ; GFC vise/Unclamp
      OUT     B55
10234 LD      M1002  ; GFC HomeEnd BothOn Fault
      ANI     M608  ; Posn.   Completion
      OR      X53  ; GFC HomePositio OK
      OUT     B56
10238 LD      M1003
      OR      Y8  ; Ax#1 Forward rotation JOG start
      ANI     M608  ; Posn.   Completion
      OR      X55  ; GFC Backward End
      OUT     B57
10243 LD      Y73  ; Loading Up
      OR      X5C  ; Loading Up End  LS
      OUT     B58
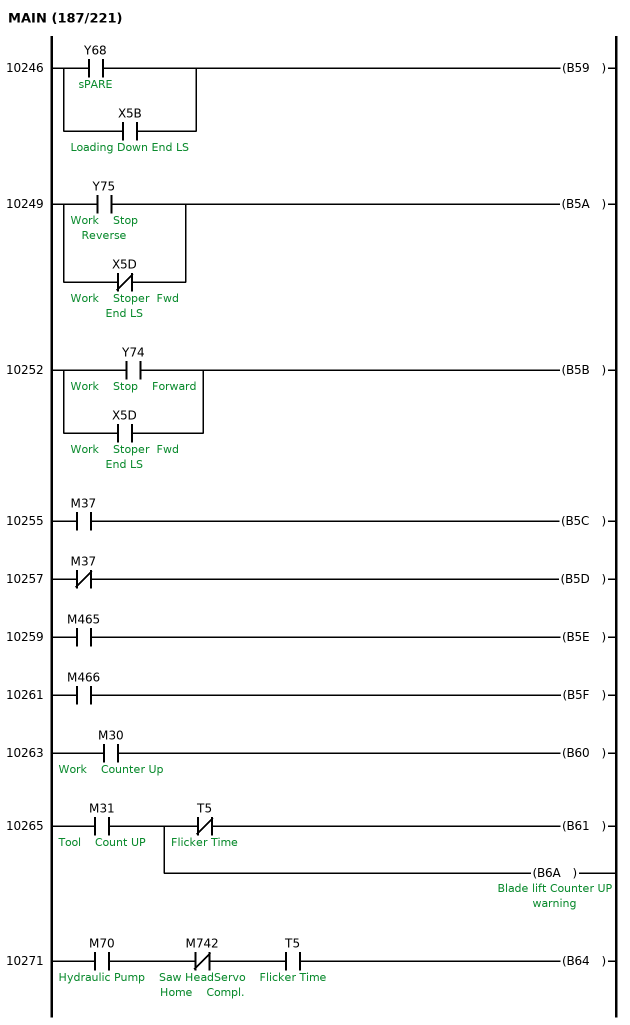
10246 LD      Y68  ; sPARE
      OR      X5B  ; Loading Down End LS
      OUT     B59
10249 LD      Y75  ; Work    Stop    Reverse
      ORI     X5D  ; Work    Stoper  Fwd End LS
      OUT     B5A
10252 LD      Y74  ; Work    Stop    Forward
      OR      X5D  ; Work    Stoper  Fwd End LS
      OUT     B5B
10255 LD      M37
      OUT     B5C
10257 LDI     M37
      OUT     B5D
10259 LD      M465
      OUT     B5E
10261 LD      M466
      OUT     B5F
10263 LD      M30  ; Work    Counter Up
      OUT     B60
10265 LD      M31  ; Tool    Count UP
      MPS
      ANI     T5  ; Flicker Time
      OUT     B61
      MPP
      OUT     B6A  ; Blade lift Counter UP warning
10271 LD      M70  ; Hydraulic Pump
      ANI     M742  ; Saw HeadServo   Home    Compl.
      AND     T5  ; Flicker Time
      OUT     B64
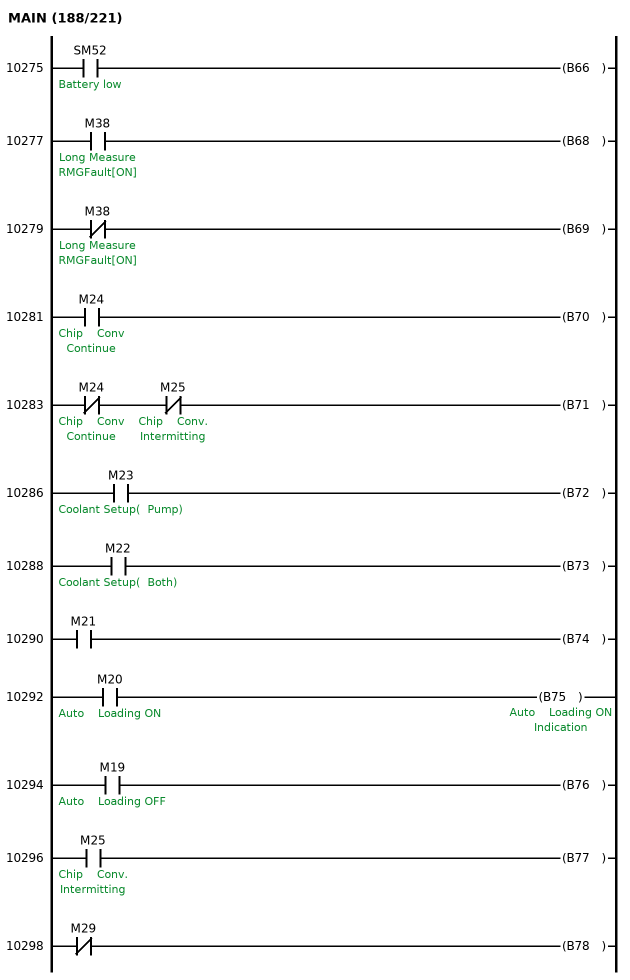
10275 LD      SM52  ; Battery low
      OUT     B66
10277 LD      M38  ; Long Measure RMGFault[ON]
      OUT     B68
10279 LDI     M38  ; Long Measure RMGFault[ON]
      OUT     B69
10281 LD      M24  ; Chip    Conv    Continue
      OUT     B70
10283 LDI     M24  ; Chip    Conv    Continue
      ANI     M25  ; Chip    Conv.   Intermitting
      OUT     B71
10286 LD      M23  ; Coolant Setup(  Pump)
      OUT     B72
10288 LD      M22  ; Coolant Setup(  Both)
      OUT     B73
10290 LD      M21
      OUT     B74
10292 LD      M20  ; Auto    Loading ON
      OUT     B75  ; Auto    Loading ON Indication
10294 LD      M19  ; Auto    Loading OFF
      OUT     B76
10296 LD      M25  ; Chip    Conv.   Intermitting
      OUT     B77
10298 LDI     M29
      OUT     B78
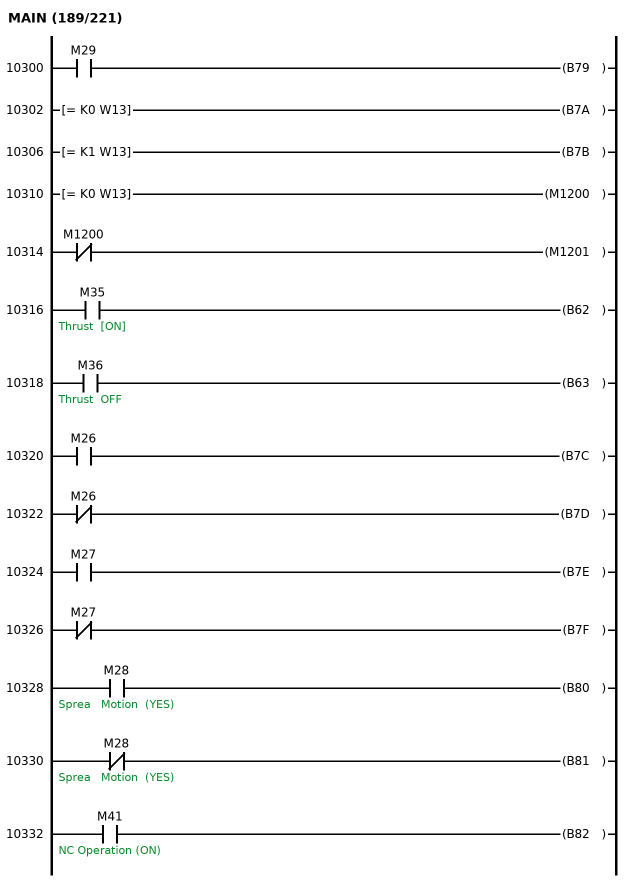
10300 LD      M29
      OUT     B79
10302 LD=     K0 W13
      OUT     B7A
10306 LD=     K1 W13
      OUT     B7B
10310 LD=     K0 W13
      OUT     M1200
10314 LDI     M1200
      OUT     M1201
10316 LD      M35  ; Thrust  [ON]
      OUT     B62
10318 LD      M36  ; Thrust  OFF
      OUT     B63
10320 LD      M26
      OUT     B7C
10322 LDI     M26
      OUT     B7D
10324 LD      M27
      OUT     B7E
10326 LDI     M27
      OUT     B7F
10328 LD      M28  ; Sprea   Motion  (YES)
      OUT     B80
10330 LDI     M28  ; Sprea   Motion  (YES)
      OUT     B81
10332 LD      M41  ; NC Operation (ON)
      OUT     B82
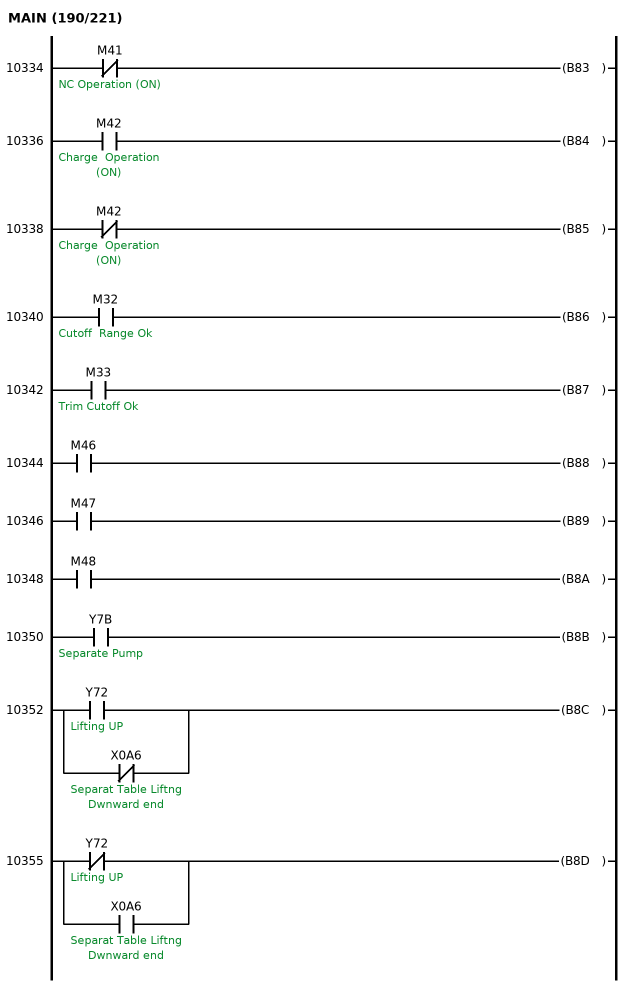
10334 LDI     M41  ; NC Operation (ON)
      OUT     B83
10336 LD      M42  ; Charge  Operation (ON)
      OUT     B84
10338 LDI     M42  ; Charge  Operation (ON)
      OUT     B85
10340 LD      M32  ; Cutoff  Range Ok
      OUT     B86
10342 LD      M33  ; Trim Cutoff Ok
      OUT     B87
10344 LD      M46
      OUT     B88
10346 LD      M47
      OUT     B89
10348 LD      M48
      OUT     B8A
10350 LD      Y7B  ; Separate Pump
      OUT     B8B
10352 LD      Y72  ; Lifting UP
      ORI     X0A6  ; Separat Table Liftng Dwnward end
      OUT     B8C
10355 LDI     Y72  ; Lifting UP
      OR      X0A6  ; Separat Table Liftng Dwnward end
      OUT     B8D
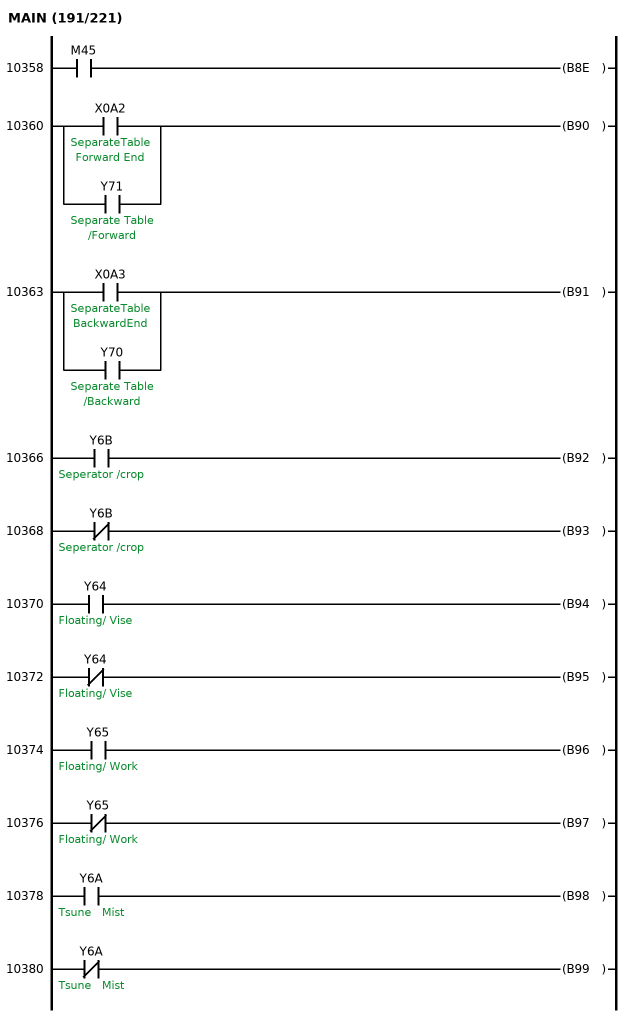
10358 LD      M45
      OUT     B8E
10360 LD      X0A2  ; SeparateTable   Forward End
      OR      Y71  ; Separate Table /Forward
      OUT     B90
10363 LD      X0A3  ; SeparateTable   BackwardEnd
      OR      Y70  ; Separate Table /Backward
      OUT     B91
10366 LD      Y6B  ; Seperator /crop
      OUT     B92
10368 LDI     Y6B  ; Seperator /crop
      OUT     B93
10370 LD      Y64  ; Floating/ Vise
      OUT     B94
10372 LDI     Y64  ; Floating/ Vise
      OUT     B95
10374 LD      Y65  ; Floating/ Work
      OUT     B96
10376 LDI     Y65  ; Floating/ Work
      OUT     B97
10378 LD      Y6A  ; Tsune   Mist
      OUT     B98
10380 LDI     Y6A  ; Tsune   Mist
      OUT     B99
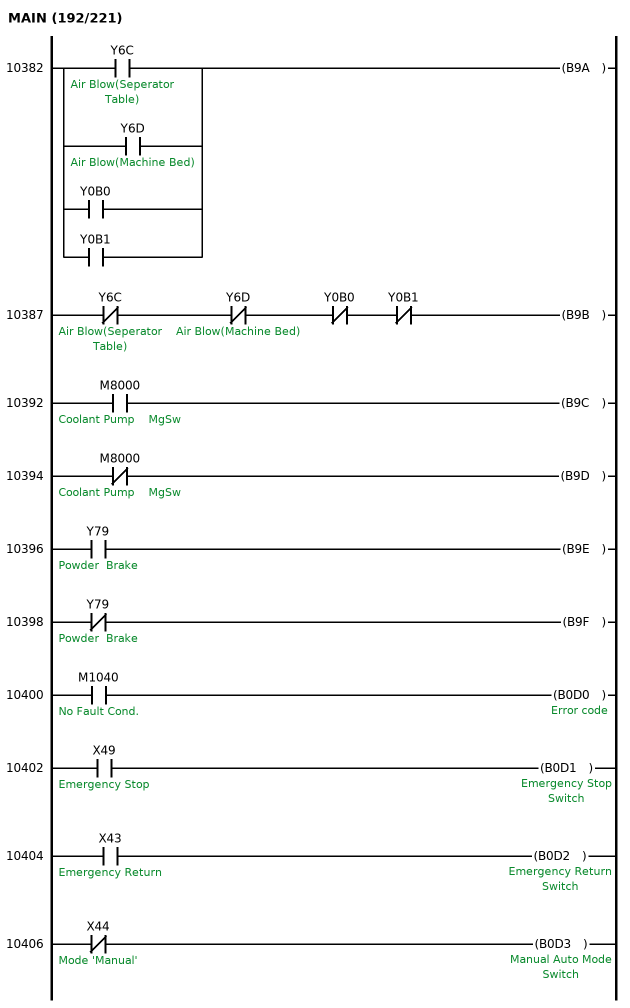
10382 LD      Y6C  ; Air Blow(Seperator Table)
      OR      Y6D  ; Air Blow(Machine Bed)
      OR      Y0B0
      OR      Y0B1
      OUT     B9A
10387 LDI     Y6C  ; Air Blow(Seperator Table)
      ANI     Y6D  ; Air Blow(Machine Bed)
      ANI     Y0B0
      ANI     Y0B1
      OUT     B9B
10392 LD      M8000  ; Coolant Pump    MgSw
      OUT     B9C
10394 LDI     M8000  ; Coolant Pump    MgSw
      OUT     B9D
10396 LD      Y79  ; Powder  Brake
      OUT     B9E
10398 LDI     Y79  ; Powder  Brake
      OUT     B9F
10400 LD      M1040  ; No Fault Cond.
      OUT     B0D0  ; Error code
10402 LD      X49  ; Emergency Stop
      OUT     B0D1  ; Emergency Stop Switch
10404 LD      X43  ; Emergency Return
      OUT     B0D2  ; Emergency Return Switch
10406 LDI     X44  ; Mode 'Manual'
      OUT     B0D3  ; Manual Auto Mode Switch
